// TwinCAT 3 PLC project EngineControlSystem
// ProgramVersion: 3.1.4023.0
// libraries:
//   Tc2_Standard, * (Beckhoff Automation GmbH)
//   Tc2_System, * (Beckhoff Automation GmbH)
//   Tc3_Module, * (Beckhoff Automation GmbH)
//   VisuSymbols,3.5.10.0,System
// project tree:
//   DUTs/ E_RotationDirection.TcDUT, ST_Inputs.TcDUT, ST_Outputs.TcDUT
//   / GlobalTextList.TcGTLO, PlcTask.TcTTO, Visualization Manager.TcVMO (not stored)
//   GVLs/ GVL_Params.TcGVL
//   OLD/ CAN_Example.TcPOU, FB_Encoder_Old1.TcPOU, FB_Encoder_Old2.TcPOU, FB_Encoder_V2.TcPOU, FB_ENCODER_V3.TcPOU, FB_HomingTimer.TcPOU, F_CounterNegativeOverflow.TcPOU (not stored), F_GenerateCANMessage.TcPOU, F_Homing.TcPOU, F_MechToEl.TcPOU, F_VoltageToWord.TcPOU, GVL_Constants.TcGVL, GVL_Measurements.TcGVL
//   POUs/ FB_Controller.TcPOU, FB_CANMessageHandler.TcPOU, FB_Encoder.TcPOU, F_AnalogIntToVoltage.TcPOU, F_VoltageToCurrentConvert.TcPOU, MAIN.TcPOU
//   VISUs/ Visualization.TcVIS
// real-time tasks:
//   TASK PlcTask: cycle T#100us, priority 1, ADS port 350
// I/O:
//   DEVICE Device 2 (EtherCAT), AmsNetId 157.24.88.195.3.1
//     Term 8 (EK1100) [EK1100 EtherCAT Coupler (2A E-Bus)]
//       Term 9 (EL5101-0010) [EL5101-0010 1Ch. Inc. Encoder 5V (20 million increments/s)]
//       Term 10 (EL3702) [EL3702 2Ch. Ana. Input +/-10V, DIFF, Oversample]
//       Term 11 (EL3702) [EL3702 2Ch. Ana. Input +/-10V, DIFF, Oversample]
//       Term 11 (EL6751) [EL6751 CANopen Master]
//       Term 12 (EL9011) [EL9011 End Terminal]
//   DEVICE Device 1 (COM Port)
//   DEVICE Device 3 (EL6751), AmsNetId 157.24.88.195.4.1
//     Zybo (CAN Interface)
// variable links:
//   EngineControlSystem/EngineControlSystem Instance <-> Device 2 (EtherCAT)/Term 8 (EK1100)/Term 10 (EL3702)
//     PlcTask Inputs/MAIN.stInputs.nEL3702Ch1_In <-> Ch1 Sample 0/Ch1 Value
//     PlcTask Inputs/MAIN.stInputs.nEL3702Ch2_In <-> Ch2 Sample 0/Ch2 Value
//   EngineControlSystem/EngineControlSystem Instance <-> Device 2 (EtherCAT)/Term 8 (EK1100)/Term 11 (EL3702)
//     PlcTask Inputs/MAIN.stInputs.nEL3702Ch3_In <-> Ch1 Sample 0/Ch1 Value
//   EngineControlSystem/EngineControlSystem Instance <-> Device 2 (EtherCAT)/Term 8 (EK1100)/Term 9 (EL5101-0010)
//     PlcTask Inputs/MAIN.stInputs.bEL5101_CounterSet <-> ENC Status compact/Status/Set counter done
//     PlcTask Inputs/MAIN.stInputs.bEL5101_LatchValid <-> ENC Status compact/Status/Latch C valid
//     PlcTask Inputs/MAIN.stInputs.nEL5101_Counter <-> ENC Status compact/Counter value
//     PlcTask Inputs/MAIN.stInputs.nEL5101_Frequency <-> ENC Frequency/Frequency value
//     PlcTask Inputs/MAIN.stInputs.nEL5101_LatchValue <-> ENC Status compact/Latch value
//     PlcTask Outputs/MAIN.stOutputs.bEL5101_EnabledLatch <-> ENC Control compact/Control/Enable latch C
//     PlcTask Outputs/MAIN.stOutputs.bEL5101_SetCounter <-> ENC Control compact/Control/Set counter
//   EngineControlSystem/EngineControlSystem Instance <-> Device 3 (EL6751)/Zybo (CAN Interface)
//     PlcTask Inputs/MAIN.stInputs.Inputs <-> Inputs/RxQueue
//     PlcTask Outputs/MAIN.stOutputs.Outputs <-> Outputs/TxQueue
//   EngineControlSystem/EngineControlSystem Instance <-> TcCOM Objects/Object2 (controller_21_1_2022)
//     PlcTask Inputs/MAIN.stInputs.fAlpha_U <-> Output/U_alpha_beta[0]
//     PlcTask Inputs/MAIN.stInputs.fBeta_U <-> Output/U_alpha_beta[1]
//     PlcTask Inputs/MAIN.stInputs.iD <-> Output/I_dq[0]
//     PlcTask Inputs/MAIN.stInputs.iQ <-> Output/I_dq[1]
//     PlcTask Outputs/MAIN.stOutputs.fControlEnable <-> Input/enable
//     PlcTask Outputs/MAIN.stOutputs.fIa <-> Input/i_abc[0]
//     PlcTask Outputs/MAIN.stOutputs.fIb <-> Input/i_abc[1]
//     PlcTask Outputs/MAIN.stOutputs.fIc <-> Input/i_abc[2]
//     PlcTask Outputs/MAIN.stOutputs.fTheta <-> Input/theta_m
//     PlcTask Outputs/MAIN.stOutputs.fWmech <-> Input/w_actual_rad_m
//     PlcTask Outputs/MAIN.stOutputs.fWref <-> Input/w_ref_rpm

CONFIGURATION EngineControlSystem
    RESOURCE PLC ON TwinCAT3
        TASK PlcTask(INTERVAL := T#100us, PRIORITY := 1);
        PROGRAM MAIN WITH PlcTask : MAIN;
    END_RESOURCE
END_CONFIGURATION

// ---- DUTs/E_RotationDirection.TcDUT
{attribute 'qualified_only'}
{attribute 'strict'}
TYPE E_RotationDirection :
(
	NONE,
	EDGE_DETECTED
);
END_TYPE

// ---- DUTs/ST_Inputs.TcDUT
TYPE ST_Inputs :
STRUCT
	// CAN
	Inputs 				AT %I*	: CANRXQUEUESTRUCT_N_1;
	
	// IO
	nEL3702Ch1_In 		AT %I*	: INT;
	nEL3702Ch2_In 		AT %I*	: INT;
	nEL3702Ch3_In 		AT %I*	: INT;
	
	// Encoder
	nEL5101_Counter 	AT %I*	: UINT;
	bEL5101_CounterSet	AT %I*	: BIT;
	nEL5101_LatchValue	AT %I*	: UINT;
	nEL5101_Frequency	AT %I*	: UDINT;
	bEL5101_LatchValid	AT %I*	: BIT;
	
	// From controller
	fAlpha_U, fBeta_U	AT %I*	: LREAL;
	iQ, iD				AT %I*	: LREAL;
END_STRUCT
END_TYPE

// ---- DUTs/ST_Outputs.TcDUT
TYPE ST_Outputs :
STRUCT
	// To controller
	fWref 					AT %Q*				: LREAL;
	fWmech					AT %Q* 				: LREAL;
	fIa, fIb, fIc 			AT %Q*				: LREAL;
	fTheta	 				AT %Q* 				: LREAL;
	fControlEnable 			AT %Q*				: LREAL;
	
	// CAN
	Outputs					AT %Q*				: CANTXQUEUESTRUCT_N_1;
	
	// Encoder
	nEL5101_SetCounterValue AT %Q*				: UINT;
	bEL5101_SetCounter		AT %Q*				: BIT;
	bEL5101_EnabledLatch	AT %Q*				: BIT;
END_STRUCT
END_TYPE

// ---- GVLs/GVL_Params.TcGVL
VAR_GLOBAL CONSTANT
	SS_INITIALIZE: SINT := 0;
	SS_STEP: SINT := 1;
END_VAR

// ---- OLD/GVL_Constants.TcGVL
{attribute 'qualified_only'}
VAR_GLOBAL CONSTANT
	PI 					: REAL 	:= 3.141592654;
	SPEED_CALC_Cycle 	: INT 	:= 100; 			// in microseconds
	NUMBER_OF_POLEPAIRS : UINT 	:= 5;
	PULSES_PER_REV 		: UINT 	:= 4096*4;
END_VAR

// ---- OLD/GVL_Measurements.TcGVL
{attribute 'qualified_only'}
VAR_GLOBAL
	COUNTER_VALUE		: UINT;
	COUNTER_OFFSET    	: UINT := 0;
	homing_done_encoder	: BOOL;
END_VAR

// ---- POUs/MAIN.TcPOU
PROGRAM MAIN
VAR
	// To controller
	bInit									: BOOL;
	fWRefPrep								: LREAL;
	
	fThetaOl								: REAL;
	
	fVa, fVb								: REAL;
	
	bZeroingDone							: BOOL;
	tpIdRun									: TP;
	tpZeroingWaitTime						: TP;
	tZeroingWaitTime						: TIME := T#1S;
	tIdTime									: TIME := T#5S;
	fElZeroAngle							: LREAL;
	
	bControlEnable							: BOOL;
	bStartHoming							: BOOL;
	bOpenLoop 								: BOOL;
	bHomingDone 							: BOOL;
	fHomingVa								: REAL := 0.5;
	fHomingVb								: REAL := 0;
	
	fbCAN_MessageHandler					: FB_CANMessageHandler();
	fbEncoder								: FB_Encoder();
	
	fbController							: FB_Controller();
	
	stInputs								: ST_Inputs;
	stOutputs								: ST_Outputs;
END_VAR

// Calling encoder and getting outputs and giving inputs
fbEncoder(	stInputs	:= stInputs,
			stOutputs	:= stOutputs,
			fThetaMech 	=> stOutputs.fTheta,
			fOmegaMech 	=> stOutputs.fWmech
);

// Id run to zero pulse location aka latch
IF NOT bZeroingDone THEN
	stOutputs.bEL5101_EnabledLatch := TRUE;
	
		fbCAN_MessageHandler(Inputs := stInputs.Inputs, 
							Outputs := stOutputs.Outputs, 
							fVoltage_A := SIN(fThetaOl),
							fVoltage_B := COS(fThetaOl));
		
		fThetaOl := fThetaOl + 2 * LREAL_TO_REAL( PI ) / 2500;
		IF fThetaOl > 2 * PI THEN
			fThetaOl := 0;
		END_IF
	
	IF stInputs.bEL5101_LatchValid THEN
		stOutputs.nEL5101_SetCounterValue := stInputs.nEL5101_LatchValue;
		stOutputs.bEL5101_SetCounter := TRUE;
		bZeroingDone := stInputs.bEL5101_CounterSet;
		stOutputs.bEL5101_EnabledLatch := FALSE;
		bStartHoming := TRUE;
	END_IF
END_IF

tpZeroingWaitTime( IN := bStartHoming, PT := tZeroingWaitTime );

// Homing
IF bStartHoming AND NOT bHomingDone AND NOT tpZeroingWaitTime.Q THEN
	tpIdRun( IN := bStartHoming, PT := tIdTime );
	stOutputs.fControlEnable := 0;
	fbCAN_MessageHandler(Inputs := stInputs.Inputs, 
						Outputs := stOutputs.Outputs, 
						fVoltage_A := fHomingVa,
						fVoltage_B := fHomingVb);
	
	IF NOT tpIdRun.Q THEN
		fElZeroAngle := fbEncoder.fThetaMech;
		bHomingDone := TRUE;
	END_IF
END_IF

// Enabling for old controller
IF bControlEnable THEN
	stOutputs.fControlEnable := 1;
ELSE	
	stOutputs.fControlEnable := 0;
END_IF 

// Getting controller outputs and giving inputs
fbController.speedrefrpm := fWRefPrep;

fbController.anglerad := -1 * ( fbEncoder.fThetaMech - fElZeroAngle );
// Multiplying the mechanical speed with number of pole pairs gives us the electrical field rotation speed
fbController.speedmeasrad := -1 * fbEncoder.fOmegaMech * 2;

fbController.Current_abc[0] := stInputs.nEL3702Ch1_In;
fbController.Current_abc[1] := stInputs.nEL3702Ch2_In;
fbController.Current_abc[2] := stInputs.nEL3702Ch3_In;

// Controller init
IF NOT bInit THEN
	fbController( ssMethodType := SS_INITIALIZE );
	bInit := TRUE;
END_IF

// Scaling of 0.9 used because svpwm doesnt like full 1 and the scaling in controller uses 400 V which is also the saturation point
fVa := LREAL_TO_REAL(fbController.Voltageoutalphabeta[0] * 0.9);
fVb := LREAL_TO_REAL(fbController.Voltageoutalphabeta[1] * 0.9);

// Enabling controller or open loop
IF bHomingDone THEN
	IF bControlEnable THEN
		IF bInit THEN
			fbController( ssMethodType := SS_STEP );
		END_IF
		fbCAN_MessageHandler(Inputs := stInputs.Inputs, 
							Outputs := stOutputs.Outputs, 
							fVoltage_A := fVa,
							fVoltage_B := fVb);
	ELSIF bOpenLoop THEN
		fbCAN_MessageHandler(Inputs := stInputs.Inputs, 
							Outputs := stOutputs.Outputs, 
							fVoltage_A := SIN(fThetaOl),
							fVoltage_B := COS(fThetaOl));
		
		fThetaOl := fThetaOl + 2 * LREAL_TO_REAL( PI ) / 2500;
		IF fThetaOl > 2 * PI THEN
			fThetaOl := 0;
		END_IF
	END_IF
END_IF

END_PROGRAM

// ---- POUs/FB_CANMessageHandler.TcPOU
FUNCTION_BLOCK FB_CANMessageHandler
VAR_INPUT
	Outputs 	: REFERENCE TO CANTXQUEUESTRUCT_N_1; // CAN muuttujat
	Inputs 		: REFERENCE TO CANRXQUEUESTRUCT_N_1;
	
	fVoltage_A	: REAL; // Jännite A realina
	fVoltage_B	: REAL; // Jännite B realina
END_VAR
VAR
	i				: DINT;
	MessageReceived : CANQUEUE;
	MessageToSend	: CANQUEUE;
	NumberOfMessagesToSend	: UINT := 1;
	wV_a,wV_b		: WORD;
END_VAR

wV_a := M_VoltageToWord(Voltage_In := fVoltage_A);
wV_b := M_VoltageToWord(Voltage_In := fVoltage_B);

MessageToSend := M_GenerateCANMessage(cobID := 4, V_a := wV_a, V_b := wV_b);

IF Outputs.TxCounter = Inputs.TxCounter THEN
   	Outputs.TxMessages[0] := MessageToSend;
    Outputs.NoOfTxMessages := NumberOfMessagesToSend;
    Outputs.TxCounter := Outputs.TxCounter + 1;
END_IF

METHOD M_GenerateCANMessage : CANQUEUE
VAR_INPUT
	cobID	: UINT;
	V_a		: WORD;
	V_b		: WORD;
END_VAR
VAR
	i,j 		: UINT;
	Tempdata	: USINT;
	V_DWORD		: WORD;
	tempMessage : CANMESSAGE;
END_VAR

// WIP CAN Message writing.
(*
	Viestiin tulee Va ja Vb (ilmeisesti). Yksi CAN Frame on käytössä näille kahdelle muuttujalle.
	CANQUEUE Objekti on yksi CAN viesti, joka lähetetään COB ID:seen ja se sisältää 8 kpl UINT muuttujia, jotka varmaankin kirjoitetaan sarjassa, josta muodostuu se 64 bittinen CAN Frame.
	Ei kyllä ole kamalasti ideaa että missä järjestyksessä ne kirjoitetaan sinne. Eli pitäisi varmaankin testata. 
	Koodi on nyt silleensä että oletetaan että kirjoitetaan 7 -> 0. Jolloin 7:n data yksikön merkitsevin bitti on koko framen merkisevin
	Vastaavasti 0:n viimeinen bitti on koko framen viimeinen kirjoitettava bitti.
*)


M_GenerateCANMessage.cobId := cobID;

V_DWORD := V_a;
FOR j := 0 TO 1 DO // First part of frame reserved for V_a
	CASE j OF // ST is dumb language and doesnt allow looping for bit access.
		1:
			Tempdata.0 := V_DWORD.0;
			Tempdata.1 := V_DWORD.1;
			Tempdata.2 := V_DWORD.2;
			Tempdata.3 := V_DWORD.3;
			Tempdata.4 := V_DWORD.4;
			Tempdata.5 := V_DWORD.5;
			Tempdata.6 := V_DWORD.6;
			Tempdata.7 := V_DWORD.7;
			
		0:
			Tempdata.0 := V_DWORD.8;
			Tempdata.1 := V_DWORD.9;
			Tempdata.2 := V_DWORD.10;
			Tempdata.3 := V_DWORD.11;
			Tempdata.4 := V_DWORD.12;
			Tempdata.5 := V_DWORD.13;
			Tempdata.6 := V_DWORD.14;
			Tempdata.7 := V_DWORD.15;
	ELSE
		RETURN;
	END_CASE
	M_GenerateCANMessage.data[j] := Tempdata;
END_FOR

V_DWORD := V_b;
FOR j := 2 TO 3 DO // Second part is reserved for V_b
	CASE j OF // ST is dumb language and doesnt allow looping for bit access.
		3:
			Tempdata.0 := V_DWORD.0;
			Tempdata.1 := V_DWORD.1;
			Tempdata.2 := V_DWORD.2;
			Tempdata.3 := V_DWORD.3;
			Tempdata.4 := V_DWORD.4;
			Tempdata.5 := V_DWORD.5;
			Tempdata.6 := V_DWORD.6;
			Tempdata.7 := V_DWORD.7;
			
		2:
			Tempdata.0 := V_DWORD.8;
			Tempdata.1 := V_DWORD.9;
			Tempdata.2 := V_DWORD.10;
			Tempdata.3 := V_DWORD.11;
			Tempdata.4 := V_DWORD.12;
			Tempdata.5 := V_DWORD.13;
			Tempdata.6 := V_DWORD.14;
			Tempdata.7 := V_DWORD.15;
	ELSE
		RETURN;
	END_CASE
	M_GenerateCANMessage.data[j] := Tempdata;
END_FOR
END_METHOD

METHOD M_VoltageToWord : WORD
VAR_INPUT
	Voltage_In			: REAL; // Voltage input
END_VAR
VAR
	VoltageMultiplier	: REAL;
	MaxWordValue		: REAL := 16#FFFF;
	Voltage_High_Value 	: REAL := 0.866;
	Voltage_Low_Value	: REAL := -0.866;
END_VAR
// Check that voltage value is between min and max value.
IF Voltage_In > Voltage_High_Value THEN
	Voltage_In := Voltage_High_Value;
ELSIF Voltage_In < Voltage_Low_Value THEN
	Voltage_In := Voltage_Low_Value;
END_IF

VoltageMultiplier := (Voltage_In-Voltage_Low_Value)/(Voltage_High_Value-Voltage_Low_Value);

M_VoltageToWord := UINT_TO_WORD(REAL_TO_UINT(VoltageMultiplier*MaxWordValue));
END_METHOD

END_FUNCTION_BLOCK

// ---- POUs/FB_Encoder.TcPOU
FUNCTION_BLOCK FB_Encoder
VAR_INPUT
	stInputs				: REFERENCE TO ST_Inputs;
	stOutputs				: REFERENCE TO ST_Outputs;
END_VAR
VAR_OUTPUT
	fThetaMech				: LREAL;
	fOmegaMech				: LREAL;
END_VAR
VAR
	bUseLatch				: BOOL;
	bInit					: BOOL;
	fOmegaMechNoDirection	: LREAL := 0.0; // No rotation direction
	fRotationDirection		: LREAL := 0.0;
	fPpr					: LREAL := 4096;
	fFreqScale				: LREAL := 0.01;
	f16bitMax				: LREAL := 65535;
	nCounter				: UINT;
	fTheta					: LREAL := 0.0;
	fThetaPrev				: LREAL := 0.0;
	nThetaDelta				: LREAL := 0.0;
	nThetaDeltaPrev			: LREAL := 0.0;
END_VAR



// Angle calculation
nCounter		:= stInputs.nEL5101_Counter * 4;
fThetaPrev 		:= fTheta;
fTheta	:= ( 2.0 * PI ) - ( UINT_TO_LREAL( nCounter ) / f16bitMax * 2.0 * PI ); // Counter is divided by max value of UINT times two because one circle is 2pi


// Rotation direction calculation
IF bUseLatch THEN
	stOutputs.bEL5101_EnabledLatch := TRUE;
	
	IF stInputs.nEL5101_LatchValue < stInputs.nEL5101_Counter THEN
		fRotationDirection := -1;
	ELSIF stInputs.nEL5101_LatchValue > stInputs.nEL5101_Counter THEN
		fRotationDirection := 1;
	END_IF
	
	stOutputs.bEL5101_EnabledLatch := FALSE;
	
ELSE
	nThetaDeltaPrev := nThetaDelta;
	nThetaDelta		:= fTheta - fThetaPrev;
	
	IF nThetaDelta < 0 AND nThetaDeltaPrev < 0 THEN
		fRotationDirection := 1;
	ELSIF  nThetaDelta > 0 AND nThetaDeltaPrev > 0  THEN
			fRotationDirection := -1;
	END_IF
END_IF

// Angle speed calculation
fOmegaMechNoDirection := 2.0 * PI * ( UDINT_TO_LREAL( stInputs.nEL5101_Frequency ) / fPpr * fFreqScale );

// Outputs
fThetaMech	:= fTheta;
fOmegaMech 	:= fRotationDirection * fOmegaMechNoDirection;

END_FUNCTION_BLOCK

// ---- POUs/FB_Controller.TcPOU
FUNCTION_BLOCK FB_Controller
VAR_INPUT
	ssMethodType: SINT;
	speedrefrpm: LREAL;
	Current_abc: ARRAY[0..2] OF LREAL;
	speedmeasrad: LREAL;
	anglerad: LREAL;
END_VAR
VAR_OUTPUT
	Voltageoutalphabeta: ARRAY[0..1] OF LREAL;
	Electrictorguecommand: LREAL;
	Currentmeasalphabeta: ARRAY[0..1] OF LREAL;
	Currentmeasdq: ARRAY[0..1] OF LREAL;
	Currentcommanddq: ARRAY[0..1] OF LREAL;
	Voltagecommanddq: ARRAY[0..1] OF LREAL;
	Voltagecommandalphabeta: ARRAY[0..1] OF LREAL;
END_VAR
VAR
	rtb_IntegralGain: LREAL;
	rtb_DeadZone: LREAL;
	rtb_DeadZone_p: LREAL;
	rtb_idref: LREAL;
	rtb_Gain3: LREAL;
	rtb_IntegralGain_p: LREAL;
	rtb_Gain4: LREAL;
	rtb_Fcn: LREAL;
	rtb_Integrator_k: LREAL;
	rtb_Fcn1: LREAL;
	rtb_iqref: LREAL;
	rtb_IntegralGain_h: LREAL;
	rtb_DeadZone_c: LREAL;
	rtb_Saturation: LREAL;
	rtb_Switch2: SINT;
	rtb_Switch1: SINT;
	rtb_Saturation_h_idx_0: LREAL;
	rtb_Saturation_h_idx_1: LREAL;
	temp1: LREAL;
	Gain3: LREAL;
	Integrator_DSTATE: LREAL;
	Integrator_DSTATE_c: LREAL;
	Integrator_DSTATE_m: LREAL;
	Gain2: LREAL;
	Sqrt2: LREAL;
	Gain4: LREAL;
END_VAR



CASE ssMethodType OF
    SS_INITIALIZE: 
        (* SystemInitialize for Atomic SubSystem: '<Root>/Controller_subsystem_29112022' *)
        (* InitializeConditions for DiscreteIntegrator: '<S145>/Integrator' *)
        Integrator_DSTATE := 0.0;
        (* InitializeConditions for DiscreteIntegrator: '<S43>/Integrator' *)
        Integrator_DSTATE_c := 0.0;
        (* InitializeConditions for DiscreteIntegrator: '<S93>/Integrator' *)
        Integrator_DSTATE_m := 0.0;
        (* End of SystemInitialize for SubSystem: '<Root>/Controller_subsystem_29112022' *)
        

        (* ConstCode for Atomic SubSystem: '<Root>/Controller_subsystem_29112022' *)
        (* ConstCode for Gain: '<S3>/Gain2' incorporates:
         *  Constant: '<S3>/Constant' *)
        Gain2 := 2.1427199999999997;
        (* ConstCode for Sqrt: '<S3>/Sqrt2' incorporates:
         *  Constant: '<S3>/Constant1' *)
        Sqrt2 := 1.4142135623730951;
        (* ConstCode for Gain: '<S3>/Gain3' *)
        Gain3 := 0.44739 * Sqrt2;
        (* ConstCode for Gain: '<S3>/Gain4' incorporates:
         *  Constant: '<S3>/Constant2' *)
        Gain4 := 2.1427199999999997;
        (* End of ConstCode for SubSystem: '<Root>/Controller_subsystem_29112022' *)
    SS_STEP: 
        (* Outputs for Atomic SubSystem: '<Root>/Controller_subsystem_29112022' *)
        (* Sum: '<S4>/Add1' incorporates:
         *  Gain: '<S1>/toRad' *)
        rtb_IntegralGain := (0.10471975511965977 * speedrefrpm) - speedmeasrad;
        (* Sum: '<S154>/Sum' incorporates:
         *  DiscreteIntegrator: '<S145>/Integrator'
         *  Gain: '<S150>/Proportional Gain' *)
        rtb_DeadZone := (0.1 * rtb_IntegralGain) + Integrator_DSTATE;
        (* Saturate: '<S152>/Saturation' *)

        IF rtb_DeadZone > 7.0 THEN 
            rtb_DeadZone_p := 7.0;
        ELSIF rtb_DeadZone >= -7.0 THEN 
            rtb_DeadZone_p := rtb_DeadZone;
        ELSE 
            rtb_DeadZone_p := -7.0;
        END_IF;

        (* End of Saturate: '<S152>/Saturation' *)
        

        (* Switch: '<S4>/Switch' incorporates:
         *  Constant: '<S4>/Constant3' *)

        IF rtb_DeadZone_p <> 0.0 THEN 
            Electrictorguecommand := rtb_DeadZone_p;
        ELSE 
            Electrictorguecommand := 0.01;
        END_IF;

        (* End of Switch: '<S4>/Switch' *)
        

        (* Product: '<S3>/Divide1' incorporates:
         *  Abs: '<S3>/Abs'
         *  Gain: '<S3>/Gain1'
         *  Product: '<S3>/Divide'
         *  Sqrt: '<S3>/Sqrt1' *)
        temp1 := ABS(Electrictorguecommand);
        rtb_idref := SQRT((0.1615435812 * temp1) / Gain2) / Gain3;
        (* Gain: '<S5>/Gain3' incorporates:
         *  Gain: '<S5>/Gain1'
         *  Gain: '<S5>/Gain2'
         *  Sum: '<S5>/Sum' *)
        rtb_Gain3 := (((-0.5 * Current_abc[1]) + Current_abc[0]) + (-0.5 * Current_abc[2])) * 0.66666666666666663;
        (* Gain: '<S5>/Gain4' incorporates:
         *  Gain: '<S5>/Gain6'
         *  Gain: '<S5>/Gain7'
         *  Sum: '<S5>/Sum1' *)
        rtb_Gain4 := ((0.8660254037844386 * Current_abc[1]) + (-0.8660254037844386 * Current_abc[2])) * 0.66666666666666663;
        (* Fcn: '<S6>/Fcn' incorporates:
         *  Fcn: '<S6>/Fcn1'
         *  Fcn: '<S7>/Fcn'
         *  Fcn: '<S7>/Fcn1' *)
        rtb_Saturation_h_idx_0 := SIN(anglerad);
        rtb_Saturation_h_idx_1 := COS(anglerad);
        rtb_Fcn := (rtb_Gain3 * rtb_Saturation_h_idx_1) + (rtb_Gain4 * rtb_Saturation_h_idx_0);
        (* Sum: '<S2>/Add' *)
        rtb_IntegralGain_p := rtb_idref - rtb_Fcn;
        (* Sum: '<S52>/Sum' incorporates:
         *  DiscreteIntegrator: '<S43>/Integrator'
         *  Gain: '<S48>/Proportional Gain' *)
        rtb_DeadZone_p := (2.0 * rtb_IntegralGain_p) + Integrator_DSTATE_c;
        (* Saturate: '<S50>/Saturation' *)

        IF rtb_DeadZone_p > 400.0 THEN 
            rtb_Integrator_k := 400.0;
        ELSIF rtb_DeadZone_p >= -400.0 THEN 
            rtb_Integrator_k := rtb_DeadZone_p;
        ELSE 
            rtb_Integrator_k := -400.0;
        END_IF;

        (* End of Saturate: '<S50>/Saturation' *)
        

        (* Fcn: '<S6>/Fcn1' *)
        rtb_Fcn1 := (( -rtb_Gain3) * rtb_Saturation_h_idx_0) + (rtb_Gain4 * rtb_Saturation_h_idx_1);
        (* Product: '<S3>/Divide2' incorporates:
         *  Gain: '<S3>/Gain5'
         *  Product: '<S3>/Multiply' *)
        rtb_iqref := (2.0 * Electrictorguecommand) / (Gain4 * rtb_idref);
        (* Sum: '<S2>/Add1' *)
        rtb_IntegralGain_h := rtb_iqref - rtb_Fcn1;
        (* Sum: '<S2>/Add2' incorporates:
         *  Gain: '<S2>/Gain'
         *  Product: '<S2>/Product' *)
        rtb_Integrator_k := rtb_Integrator_k - ((0.09027 * rtb_Fcn1) * speedmeasrad);
        (* Sum: '<S102>/Sum' incorporates:
         *  DiscreteIntegrator: '<S93>/Integrator'
         *  Gain: '<S98>/Proportional Gain' *)
        rtb_DeadZone_c := (2.0 * rtb_IntegralGain_h) + Integrator_DSTATE_m;
        (* Saturate: '<S100>/Saturation' *)

        IF rtb_DeadZone_c > 400.0 THEN 
            rtb_Saturation := 400.0;
        ELSIF rtb_DeadZone_c >= -400.0 THEN 
            rtb_Saturation := rtb_DeadZone_c;
        ELSE 
            rtb_Saturation := -400.0;
        END_IF;

        (* End of Saturate: '<S100>/Saturation' *)
        

        (* Sum: '<S2>/Add3' incorporates:
         *  Gain: '<S2>/Gain1'
         *  Product: '<S2>/Product1' *)
        rtb_Saturation := ((0.44739 * rtb_Fcn) * speedmeasrad) + rtb_Saturation;
        (* Saturate: '<S1>/Saturation' incorporates:
         *  Fcn: '<S7>/Fcn'
         *  Fcn: '<S7>/Fcn1'
         *  Outport: '<Root>/Voltage command alpha-beta' *)
        Voltagecommandalphabeta[0] := (rtb_Integrator_k * rtb_Saturation_h_idx_1) - (rtb_Saturation * rtb_Saturation_h_idx_0);
        Voltagecommandalphabeta[1] := (rtb_Integrator_k * rtb_Saturation_h_idx_0) + (rtb_Saturation * rtb_Saturation_h_idx_1);

        IF Voltagecommandalphabeta[0] > 400.0 THEN 
            rtb_Saturation_h_idx_0 := 400.0;
        ELSIF Voltagecommandalphabeta[0] >= -400.0 THEN 
            rtb_Saturation_h_idx_0 := Voltagecommandalphabeta[0];
        ELSE 
            rtb_Saturation_h_idx_0 := -400.0;
        END_IF;


        IF Voltagecommandalphabeta[1] > 400.0 THEN 
            rtb_Saturation_h_idx_1 := 400.0;
        ELSIF Voltagecommandalphabeta[1] >= -400.0 THEN 
            rtb_Saturation_h_idx_1 := Voltagecommandalphabeta[1];
        ELSE 
            rtb_Saturation_h_idx_1 := -400.0;
        END_IF;

        (* End of Saturate: '<S1>/Saturation' *)
        

        (* DeadZone: '<S36>/DeadZone' *)

        IF rtb_DeadZone_p > 400.0 THEN 
            rtb_DeadZone_p := rtb_DeadZone_p - 400.0;
            (* Switch: '<S34>/Switch1' incorporates:
             *  Constant: '<S34>/Constant' *)
            rtb_Switch2 := 1;
        ELSE 

            IF rtb_DeadZone_p >= -400.0 THEN 
                rtb_DeadZone_p := 0.0;
            ELSE 
                rtb_DeadZone_p := rtb_DeadZone_p - -400.0;
            END_IF;

            (* Switch: '<S34>/Switch1' incorporates:
             *  Constant: '<S34>/Constant2' *)
            rtb_Switch2 := -1;
        END_IF;

        (* End of DeadZone: '<S36>/DeadZone' *)
        

        (* Gain: '<S40>/Integral Gain' *)
        rtb_IntegralGain_p := 0.2 * rtb_IntegralGain_p;
        (* Switch: '<S34>/Switch2' incorporates:
         *  Constant: '<S34>/Clamping_zero'
         *  Constant: '<S34>/Constant3'
         *  Constant: '<S34>/Constant4'
         *  RelationalOperator: '<S34>/fix for DT propagation issue1' *)

        IF rtb_IntegralGain_p > 0.0 THEN 
            rtb_Switch1 := 1;
        ELSE 
            rtb_Switch1 := -1;
        END_IF;

        (* End of Switch: '<S34>/Switch2' *)
        

        (* Switch: '<S34>/Switch' incorporates:
         *  Constant: '<S34>/Clamping_zero'
         *  Constant: '<S34>/Constant1'
         *  Logic: '<S34>/AND3'
         *  RelationalOperator: '<S34>/Equal1'
         *  RelationalOperator: '<S34>/Relational Operator' *)

        IF (rtb_DeadZone_p <> 0.0) AND (rtb_Switch2 = rtb_Switch1) THEN 
            rtb_IntegralGain_p := 0.0;
        END_IF;

        (* End of Switch: '<S34>/Switch' *)
        

        (* DeadZone: '<S86>/DeadZone' *)

        IF rtb_DeadZone_c > 400.0 THEN 
            rtb_DeadZone_c := rtb_DeadZone_c - 400.0;
            (* Switch: '<S84>/Switch1' incorporates:
             *  Constant: '<S84>/Constant' *)
            rtb_Switch1 := 1;
        ELSE 

            IF rtb_DeadZone_c >= -400.0 THEN 
                rtb_DeadZone_c := 0.0;
            ELSE 
                rtb_DeadZone_c := rtb_DeadZone_c - -400.0;
            END_IF;

            (* Switch: '<S84>/Switch1' incorporates:
             *  Constant: '<S84>/Constant2' *)
            rtb_Switch1 := -1;
        END_IF;

        (* End of DeadZone: '<S86>/DeadZone' *)
        

        (* Gain: '<S90>/Integral Gain' *)
        rtb_IntegralGain_h := 0.2 * rtb_IntegralGain_h;
        (* Switch: '<S84>/Switch2' incorporates:
         *  Constant: '<S84>/Clamping_zero'
         *  Constant: '<S84>/Constant3'
         *  Constant: '<S84>/Constant4'
         *  RelationalOperator: '<S84>/fix for DT propagation issue1' *)

        IF rtb_IntegralGain_h > 0.0 THEN 
            rtb_Switch2 := 1;
        ELSE 
            rtb_Switch2 := -1;
        END_IF;

        (* End of Switch: '<S84>/Switch2' *)
        

        (* Switch: '<S84>/Switch' incorporates:
         *  Constant: '<S84>/Clamping_zero'
         *  Constant: '<S84>/Constant1'
         *  Logic: '<S84>/AND3'
         *  RelationalOperator: '<S84>/Equal1'
         *  RelationalOperator: '<S84>/Relational Operator' *)

        IF (rtb_DeadZone_c <> 0.0) AND (rtb_Switch1 = rtb_Switch2) THEN 
            rtb_IntegralGain_h := 0.0;
        END_IF;

        (* End of Switch: '<S84>/Switch' *)
        

        (* DeadZone: '<S138>/DeadZone' *)

        IF rtb_DeadZone > 7.0 THEN 
            rtb_DeadZone := rtb_DeadZone - 7.0;
            (* Switch: '<S136>/Switch1' incorporates:
             *  Constant: '<S136>/Constant' *)
            rtb_Switch1 := 1;
        ELSE 

            IF rtb_DeadZone >= -7.0 THEN 
                rtb_DeadZone := 0.0;
            ELSE 
                rtb_DeadZone := rtb_DeadZone - -7.0;
            END_IF;

            (* Switch: '<S136>/Switch1' incorporates:
             *  Constant: '<S136>/Constant2' *)
            rtb_Switch1 := -1;
        END_IF;

        (* End of DeadZone: '<S138>/DeadZone' *)
        

        (* Gain: '<S142>/Integral Gain' *)
        rtb_IntegralGain := 0.05 * rtb_IntegralGain;
        (* Switch: '<S136>/Switch2' incorporates:
         *  Constant: '<S136>/Clamping_zero'
         *  Constant: '<S136>/Constant3'
         *  Constant: '<S136>/Constant4'
         *  RelationalOperator: '<S136>/fix for DT propagation issue1' *)

        IF rtb_IntegralGain > 0.0 THEN 
            rtb_Switch2 := 1;
        ELSE 
            rtb_Switch2 := -1;
        END_IF;

        (* End of Switch: '<S136>/Switch2' *)
        

        (* Switch: '<S136>/Switch' incorporates:
         *  Constant: '<S136>/Clamping_zero'
         *  Constant: '<S136>/Constant1'
         *  Logic: '<S136>/AND3'
         *  RelationalOperator: '<S136>/Equal1'
         *  RelationalOperator: '<S136>/Relational Operator' *)

        IF (rtb_DeadZone <> 0.0) AND (rtb_Switch1 = rtb_Switch2) THEN 
            rtb_IntegralGain := 0.0;
        END_IF;

        (* End of Switch: '<S136>/Switch' *)
        

        (* Update for DiscreteIntegrator: '<S145>/Integrator' *)
        Integrator_DSTATE := (5.0E-5 * rtb_IntegralGain) + Integrator_DSTATE;
        (* Update for DiscreteIntegrator: '<S43>/Integrator' *)
        Integrator_DSTATE_c := (5.0E-5 * rtb_IntegralGain_p) + Integrator_DSTATE_c;
        (* Update for DiscreteIntegrator: '<S93>/Integrator' *)
        Integrator_DSTATE_m := (5.0E-5 * rtb_IntegralGain_h) + Integrator_DSTATE_m;
        (* Outport: '<Root>/Voltage out alpha-beta' incorporates:
         *  Gain: '<S1>/normalize' *)
        Voltageoutalphabeta[0] := 0.0025 * rtb_Saturation_h_idx_0;
        Voltageoutalphabeta[1] := 0.0025 * rtb_Saturation_h_idx_1;
        (* End of Outputs for SubSystem: '<Root>/Controller_subsystem_29112022' *)
        

        (* Outport: '<Root>/Current meas alpha-beta' *)
        Currentmeasalphabeta[0] := rtb_Gain3;
        Currentmeasalphabeta[1] := rtb_Gain4;
        (* Outport: '<Root>/Current meas dq' *)
        Currentmeasdq[0] := rtb_Fcn;
        Currentmeasdq[1] := rtb_Fcn1;
        (* Outport: '<Root>/Current command dq' *)
        Currentcommanddq[0] := rtb_idref;
        Currentcommanddq[1] := rtb_iqref;
        (* Outport: '<Root>/Voltage command dq' *)
        Voltagecommanddq[0] := rtb_Integrator_k;
        Voltagecommanddq[1] := rtb_Saturation;
END_CASE;

END_FUNCTION_BLOCK

// ---- OLD/CAN_Example.TcPOU
FUNCTION_BLOCK CAN_Example
VAR_INPUT
END_VAR
VAR_OUTPUT
END_VAR
VAR
	fPhase1_Uptime	: DINT;
	fPhase2_Uptime	: DINT;
	fPhase3_Uptime	: DINT;
	fPhase1_Offset	: DINT;
	fPhase2_Offset	: DINT;
	fPhase3_Offset	: DINT;
END_VAR

(*
Example codes from some beckhoff PDF

Sample code: Sending messages from the PLC
if Outputs.TxCounter = Inputs.TxCounter then
          for i=0 to NumberOfMessagesToSend do
                  Outputs.TxMessage[i] = MessageToSend[i];
          End_for
          Outputs.NoOfTxMessages = NumberOfMessagesToSend;
          Outputs.TxCounter := Outputs.TxCounter + 1;
end_if


Sample code: Receiving messages from the PLC
if Outputs.RxCounter <> Inputs.RxCounter then
          for I := 0 to (Inputs.NoOfRxMessages-1) do
                   MessageReceived[i] := Inputs.RxMessage [i];
          End_for
          Outputs.RxCounter := Outputs.RxCounter+1;
end_if

*)

END_FUNCTION_BLOCK

// ---- OLD/FB_Encoder_Old1.TcPOU
FUNCTION_BLOCK FB_Encoder_Old1
VAR_OUTPUT
	THETA 					: REAL;
	THETA_EL 				: REAL;
	OMEGA					: REAL;
END_VAR
VAR
	OMEGA_raw				: REAL;
	OMEGA_filtered			: REAL;
	Omega_prev				: REAL;
	THETA_rads				: REAL;
	THETA_prev_rads			: REAL;
	
	THETA_PREV 				: REAL 	:= 0;
	T_S 					: REAL 	:= 0.0001;
	OVERFLOW_SET 			: BOOL 	:= FALSE;
	UNDERFLOW_SET 			: BOOL 	:= FALSE;

	UNDERFLOW_VALUE 		: UINT 	:= 0;
	OVERFLOW_VALUE 			: UINT 	:= 4096*4; //65535;
	DOWNCOUNT_VALUE 		: UINT 	:= 1003;
	UPCOUNT_VALUE 			: UINT 	:= DOWNCOUNT_VALUE + (Constants.PULSES_PER_REV - 1);
	
	INIT_DONE 				: BOOL 	:= FALSE;
	
	COUNTER_VALUE			: UINT;
	I 						: INT 	:= 0;
	COUNTER_VALUE_PREV 		: UINT 	:= Measurements.COUNTER_VALUE;
	COUNTER_OUT 			: UINT 	:= 0;
	FIRSTCYCLE_DONE 		: BOOL 	:= FALSE;
	CLOCKWISE				: BOOL;
	COUNTERCLOCKWISE		: BOOL;
	PLUSONEPULSE 			: BOOL;
	PLUSTWOPULSES 			: BOOL;
	PLUSTHREEPULSES 		: BOOL;
	
	THETA_EST_TOT 			: REAL;
	THETA_EST_TOT_OLD		: REAL	:=0.0;
	THETA_ERR_FAST			: REAL;
	THETA_ERR_HYS			: REAL	:= 0.1;	//0.1
	OMEGA_FAST 				: REAL;
	OMEGA_EST_TOT 			: REAL;
	Ts_EST 					: REAL 	:=1E-4;	//1E-2
	THETA_EST_FAST 			: REAL;
	THETA_EST_FAST_OLD 		: REAL;
	GAIN_EST 				: REAL 	:=20; 	//1
	
	THETA_n 				: REAL; 
	DELTA_THETA_n0 			: REAL :=0.0;
	DELTA_THETA_n1 			: REAL :=0.0; 
	DELTA_THETA 			: REAL;
	temp					: REAL; 
END_VAR

// counter resetointi. kirjoita arvo enc control compact/control/set counter value ja rising edge /control/set counter


COUNTER_VALUE := Measurements.COUNTER_VALUE;

//Init procedure
IF FIRSTCYCLE_DONE = FALSE THEN
(*	STARTING_VALUE := COUNTER_VALUE;
	UP_VALUE := STARTING_VALUE + PULSES_PER_REV;
	DOWN_VALUE := STARTING_VALUE - PULSES_PER_REV;
*)	FIRSTCYCLE_DONE := TRUE;
END_IF

//End of init procedure

//Rotation direction estimation											//ADDED ROTATION  DIRECTION ESTIMATION - FEDOR POLUNIN 07 06 17

	IF (COUNTER_VALUE < COUNTER_VALUE_PREV AND COUNTER_VALUE <= (UNDERFLOW_VALUE + 2) AND COUNTER_VALUE_PREV >= (OVERFLOW_VALUE - 2)) THEN
		CLOCKWISE := TRUE;
		COUNTERCLOCKWISE := FALSE;
	ELSIF (COUNTER_VALUE > COUNTER_VALUE_PREV AND COUNTER_VALUE_PREV <= (UNDERFLOW_VALUE + 2) AND COUNTER_VALUE >= (OVERFLOW_VALUE - 2)) THEN
		COUNTERCLOCKWISE := TRUE;
		CLOCKWISE := FALSE;
	ELSIF 	(COUNTER_VALUE > COUNTER_VALUE_PREV AND COUNTER_VALUE <> OVERFLOW_VALUE) THEN 
		CLOCKWISE := TRUE;
		COUNTERCLOCKWISE := FALSE;
	ELSIF 	(COUNTER_VALUE < COUNTER_VALUE_PREV AND COUNTER_VALUE <> UNDERFLOW_VALUE) THEN
		COUNTERCLOCKWISE := TRUE;
		CLOCKWISE := FALSE;
	END_IF

//COUNTERCLOCKWISE := TRUE;
//CLOCKWISE := TRUE;

//End of Rotation direction estimation 

// Counter value conversion from 0..65535 to DOWNCOUNT_VALUE .. UPCOUNT_VALUE (1003..2002)  		//up to 1200 rpm both directions, no pulse loss w/o load Fedor Polunin 26 06 2017

IF (COUNTER_VALUE <= (UNDERFLOW_VALUE + 2) AND COUNTER_VALUE_PREV >= (OVERFLOW_VALUE - 2)) THEN
	COUNTER_OUT := COUNTER_OUT + (COUNTER_VALUE-UNDERFLOW_VALUE) + (OVERFLOW_VALUE-COUNTER_VALUE_PREV) + 1; 	//added + 1 because otherwise when COUNTER_VALUE resets from 65535 to 0, COUNTER_OUT does not increment
ELSIF (COUNTER_VALUE >= (OVERFLOW_VALUE - 2) AND COUNTER_VALUE_PREV <= (UNDERFLOW_VALUE + 2)) THEN
	COUNTER_OUT := COUNTER_OUT - (OVERFLOW_VALUE-COUNTER_VALUE) - (COUNTER_VALUE_PREV-UNDERFLOW_VALUE) - 1;		//added - 1 because otherwise when COUNTER_VALUE resets from 0 to 65535, COUNTER_OUT does not decrement
ELSIF (COUNTER_VALUE = COUNTER_VALUE_PREV + 1) OR (COUNTER_VALUE = COUNTER_VALUE_PREV + 2) OR (COUNTER_VALUE = COUNTER_VALUE_PREV + 3)THEN			
	COUNTER_OUT := COUNTER_OUT + (COUNTER_VALUE - COUNTER_VALUE_PREV); // + 1;
ELSIF  (COUNTER_VALUE = COUNTER_VALUE_PREV - 1) OR (COUNTER_VALUE = COUNTER_VALUE_PREV - 2) OR (COUNTER_VALUE = COUNTER_VALUE_PREV - 3) THEN; 
	COUNTER_OUT := COUNTER_OUT - (COUNTER_VALUE_PREV - COUNTER_VALUE);//- 1;
END_IF

IF COUNTER_OUT < DOWNCOUNT_VALUE THEN
	COUNTER_OUT := UPCOUNT_VALUE - (DOWNCOUNT_VALUE - COUNTER_OUT) + 1;  // +1 TO PREVENT COUNTER_OUT FROM SETTING UP TO 2001 INSTEAD OF 2002 WHEN DOWNCOUNT_VALUE - COUNTER_OUT = 1
	UNDERFLOW_SET := TRUE;
	
ELSIF COUNTER_OUT > UPCOUNT_VALUE THEN
	COUNTER_OUT := DOWNCOUNT_VALUE + (COUNTER_OUT - UPCOUNT_VALUE) - 1;  //FOR THE SAME REASON
	OVERFLOW_SET := TRUE;
END_IF

(*	
	//Encoder pulses per program cycle counter														
IF (COUNTER_VALUE = COUNTER_VALUE_PREV + 1) THEN
	PLUSONEPULSE := TRUE;
	PLUSTWOPULSES := FALSE;
	PLUSTHREEPULSES := FALSE;
	
ELSIF (COUNTER_VALUE = COUNTER_VALUE_PREV + 2) THEN
	PLUSONEPULSE := FALSE;
	PLUSTWOPULSES := TRUE;
	PLUSTHREEPULSES := FALSE;
	
ELSIF (COUNTER_VALUE = COUNTER_VALUE_PREV + 3) THEN
	PLUSONEPULSE := FALSE;
	PLUSTWOPULSES := FALSE;
	PLUSTHREEPULSES := TRUE;
END_IF
*)

COUNTER_VALUE_PREV := COUNTER_VALUE;

//End of counter value conversion 

// Convert to rotor angle theta in degrees

	THETA := 360.0*INT_TO_REAL(UINT_TO_INT(COUNTER_OUT - DOWNCOUNT_VALUE))/(UPCOUNT_VALUE-DOWNCOUNT_VALUE);		// COUNTER_OUT - DOWNCOUNT_VALUE can be negative, requires INT_TO_REAL 
	IF Measurements.homing_done_encoder THEN
		THETA := 360.0*INT_TO_REAL(COUNTER_OUT - DOWNCOUNT_VALUE)/(UPCOUNT_VALUE-DOWNCOUNT_VALUE) - Measurements.theta_nolla*180/PI;		// COUNTER_OUT - DOWNCOUNT_VALUE can be negative, requires INT_TO_REAL 
		IF THETA < 0 THEN
			temp := Measurements.theta_nolla*180/PI - (360.0*INT_TO_REAL(COUNTER_OUT - DOWNCOUNT_VALUE)/(UPCOUNT_VALUE-DOWNCOUNT_VALUE));
			THETA := 2*PI - temp;
		END_IF
	END_IF
    THETA_EL := 360.0*INT_TO_REAL(((COUNTER_OUT - DOWNCOUNT_VALUE) MOD 200))/200.0;

//End of conversion to rotor angle theta in degrees

//Angular rotation speed omega estimation (in rad/s)
I := I+1;

	THETA_rads := THETA/180*PI;

IF I = Constants.SPEED_CALC_Cycle THEN															
	// Calculate angular speed
		//raw speed estimation algorithm based on backward Euler differentiation
	IF OVERFLOW_SET = TRUE AND THETA < 20 THEN								//Fedor Polunin 06.06.17 - added AND THETA < 10 to prevent this from executing if theta hasn't yet changed from 2pi to zero
		OMEGA := (THETA + (360.0 - THETA_PREV))/(T_S*Constants.SPEED_CALC_Cycle);				
	ELSIF UNDERFLOW_SET = TRUE AND THETA > 340 THEN							//Fedor Polunin 06.06.17 - added AND THETA < 10 to prevent this from executing if theta hasn't yet changed from zero to 2pi
		OMEGA := -((360.0-THETA) + THETA_PREV)/(T_S*Constants.SPEED_CALC_Cycle);					
	ELSE
		IF CLOCKWISE = TRUE AND THETA_PREV > 180 AND THETA < 180 THEN		//Fedor Polunin 06.06.17 - added                                                                                           (IF THETA_PREV > 180 AND THETA < 180 THEN) BUT NOT VALID if both directions are used (it is to ensure correct omega estimation during THETA 2pi to 0 change)
			OMEGA := (THETA + (360.0 - THETA_PREV))/(T_S*Constants.SPEED_CALC_Cycle);			//Fedor Polunin 06.06.17 - added OMEGA := (THETA + (360.0 - THETA_PREV))/(T_S*100.0);
		ELSIF  COUNTERCLOCKWISE = TRUE AND  THETA_PREV < 180 AND THETA > 180 THEN							
			OMEGA := -((360.0-THETA) + THETA_PREV)/(T_S*Constants.SPEED_CALC_Cycle);			
		ELSE																//Fedor Polunin 06.06.17 - ELSE use theta and theta_prev without modification:
			OMEGA := (THETA - THETA_PREV)/(T_S*Constants.SPEED_CALC_Cycle);
		END_IF
	END_IF	
	
	OMEGA_raw := PI*OMEGA/180.0;
	
	//end of raw speed estimation algorithm														
	
	//filtered speed estimation algorithm based on ZOH differentiation + filter + output median filtering		
	IF OVERFLOW_SET = TRUE AND THETA < 20 THEN								//Fedor Polunin 06.06.17 - added AND THETA < 10 to prevent this from executing if theta hasn't yet changed from 2pi to zero
		DELTA_THETA := (THETA_rads + (2*PI - THETA_prev_rads));		
	ELSIF UNDERFLOW_SET = TRUE AND THETA > 340 THEN							//Fedor Polunin 06.06.17 - added AND THETA < 10 to prevent this from executing if theta hasn't yet changed from zero to 2pi
		DELTA_THETA := -((2*PI-THETA_rads ) + THETA_prev_rads);				
	ELSE
		IF CLOCKWISE = TRUE AND THETA_PREV > 180 AND THETA < 180 THEN		//Fedor Polunin 06.06.17 - added                                                                                           (IF THETA_PREV > 180 AND THETA < 180 THEN) BUT NOT VALID if both directions are used (it is to ensure correct omega estimation during THETA 2pi to 0 change)
			DELTA_THETA := (THETA_rads  + (2*PI - THETA_prev_rads));				//Fedor Polunin 06.06.17 - added OMEGA := (THETA + (360.0 - THETA_PREV))/(T_S*100.0);
		ELSIF  COUNTERCLOCKWISE = TRUE AND  THETA_PREV < 180 AND THETA > 180 THEN							
			DELTA_THETA := -((2*PI-THETA_rads ) + THETA_prev_rads);	
		ELSE																//Fedor Polunin 06.06.17 - ELSE use theta and theta_prev without modification:
			DELTA_THETA := (THETA_rads  - THETA_prev_rads);	
		END_IF
	END_IF														
	
	DELTA_THETA_n0:=0.5*DELTA_THETA+ 0.5*DELTA_THETA_n1;
 	DELTA_THETA_n1:= DELTA_THETA_n0;
	OMEGA_filtered := DELTA_THETA_n0*33*104.0166/21.23 +  0.189 * Omega_prev ;	

	THETA_PREV := THETA;
	THETA_prev_rads := THETA_rads;
	OMEGA_prev:= OMEGA_filtered;
	
	//end of filtered speed estimation algorithm
	
	I := 0;

	UNDERFLOW_SET := FALSE;
	OVERFLOW_SET := FALSE;
	
	//Speed feedback signal selection
		//OMEGA:=OMEGA_raw;
		OMEGA:=OMEGA_filtered;
		//OMEGA := PI*OMEGA/180.0;
END_IF;
	
	//fast speed estimator part (filtered algorithm above is the slow part) - refer to the paper "A Low-Noise Estimator of Angular Speed and Acceleration from Shaft Encoder Measurements"
(*
	THETA_ERR_FAST:=THETA_rads-THETA_EST_TOT;
	//  limit maybe to much lower than 2pi 
	
	IF abs(THETA_ERR_FAST) > THETA_ERR_HYS THEN
		OMEGA_FAST:= GAIN_EST*THETA_ERR_FAST;
		
	ELSE
 		OMEGA_FAST:=0;

	END_IF			
	

	OMEGA_EST_TOT:= OMEGA_filtered+OMEGA_FAST;
	THETA_EST_FAST := THETA_EST_FAST_OLD+ OMEGA_EST_TOT*Ts_EST;
	THETA_EST_TOT:=THETA_EST_FAST +0.5*Ts_EST*OMEGA_filtered;
	REST:=THETA_EST_TOT;
	
	 //IF THETA_EST_TOT >= 2*pi 
	IF THETA_EST_TOT < 0 THEN
		THETA_EST_TOT_OLD :=THETA_EST_TOT_OLD+2*PI;   
		THETA_EST_TOT := 2*PI+THETA_EST_TOT;// - (0 - THETA_EST_TOT) ;  
		THETA_EST_FAST_OLD :=THETA_EST_FAST_OLD+2*PI;   
		THETA_EST_FAST:= 2*PI+THETA_EST_FAST;
		
	//UNDERFLOW_SET := TRUE;
	
	ELSIF THETA_EST_TOT > 2*PI THEN
		THETA_EST_TOT_OLD :=THETA_EST_TOT_OLD-2*PI;   ;
		THETA_EST_TOT := THETA_EST_TOT-2*PI;// - (0 - THETA_EST_TOT) ;  
		THETA_EST_FAST_OLD :=0;//THETA_EST_FAST_OLD-2*PI;   
		THETA_EST_FAST:= 0;//THETA_EST_FAST-2*PI;
		//THETA_EST_TOT := 0;// + (THETA_EST_TOT - 2*PI) ;  //FOR THE SAME REASON
	//OVERFLOW_SET := TRUE;
	END_IF
		
		THETA_EST_FAST_OLD:= THETA_EST_FAST;
		THETA_EST_TOT_OLD := THETA_EST_TOT; 
	
	//end of fast speed estimator part
*)

//End of angular rotation speed estimation

//Rotor angle theta conversion deg -> rad and limitation
THETA := PI*THETA/180.0;
THETA_EL := PI*THETA_EL/180.0;

IF THETA < 0 THEN
	THETA := 0;
ELSIF
	THETA > 2*PI THEN
	THETA := 2*PI;
END_IF

IF THETA_EL < 0 THEN
	THETA_EL := 0;
ELSIF THETA_EL > 2*PI THEN
	THETA_EL := 2*PI;
END_IF

//End of rotor angle theta conversion deg->rad and limitation

END_FUNCTION_BLOCK

// ---- OLD/FB_Encoder_Old2.TcPOU
FUNCTION_BLOCK FB_Encoder_Old2
VAR CONSTANT
	nAmountOfSamples				: UINT := 100;
	fSamplingTime					: REAL := 0.00005; // 50us
	fCounterToRotationMultiplier	: REAL := 0.25; // Multiplier that transforms the counter value back to rotation.
	fMaxCounterIncrement			: REAL := 30000;
END_VAR
VAR
	nCounterValue 					: REFERENCE TO UINT; // Reference to value that holds the encoder value
	aPositionArray					: ARRAY [0..nAmountOfSamples-1] OF UINT; // Hold those positions in array.
	nValueCount						: UINT; // Rolling number used to store positions
	nStartCount						: UINT; // Value that holds the current starting value.
END_VAR

METHOD AddPosition : BOOL

IF nValueCount < nAmountOfSamples THEN // Fill samples
	aPositionArray[nValueCount] := nCounterValue;
	nStartCount := 0;
	nValueCount := nValueCount + 1;
ELSE // When all samples are full, move starting point forward by one. Write new value.
	nStartCount := nStartCount + 1;
	IF nStartCount = nAmountOfSamples THEN
		nStartCount := 0;
	END_IF
	
	IF nStartCount = 0 THEN
		aPositionArray[nValueCount] := nCounterValue;
	ELSE
		aPositionArray[nStartCount-1] := nCounterValue;
	END_IF
	
END_IF
END_METHOD

METHOD CalculateSpeed : REAL
VAR
	i,j 				: UINT;
	nUINTMax			: REAL := 16#FFFF;
	fTempRotationValueS	: REAL;
	fTempRotationValueE : REAL;
	fTempTotalRotation	: REAL := 0.0;
	fTempRotation		: REAL := 0.0;
	fTimeDuration		: REAL;
END_VAR
IF nValueCount < nAmountOfSamples THEN
	CalculateSpeed := 0;
ELSE
	CalculateSpeed := 0;
	fTimeDuration := fSamplingTime * nAmountOfSamples;
	FOR i := 0 TO nAmountOfSamples-1 DO
		j := nStartCount + i;
		IF j > nAmountOfSamples-1 THEN
			j := j-nAmountOfSamples;
		END_IF
		fTempRotationValueS	:= UINT_TO_REAL(aPositionArray[j]);
		
		IF j = nAmountOfSamples-1 THEN // If j value is at max index.
			fTempRotationValueE	:= UINT_TO_REAL(aPositionArray[0]);
		ELSE
			fTempRotationValueE	:= UINT_TO_REAL(aPositionArray[j+1]);
		END_IF
		
		fTempRotation := fTempRotationValueE - fTempRotationValueS; // The difference between starting point and the end point == Distance rotated between the cycles
		
		// Detection for counter overflow
		IF fTempRotation < -fMaxCounterIncrement THEN
			fTempRotation := fTempRotationValueE - fTempRotationValueS+nUINTMax;
		ELSIF fTempRotation > fMaxCounterIncrement THEN
			fTempRotation := fTempRotationValueE-nUINTMax - fTempRotationValueS;
		END_IF
		
		fTempTotalRotation := fTempTotalRotation + (fTempRotation * fCounterToRotationMultiplier);
	END_FOR
	CalculateSpeed := fTempTotalRotation/fTimeDuration; // Total Rotations during the measurement duration
	CalculateSpeed := CalculateSpeed * (60/fTimeDuration); // Multiplied to Rounds per minute
END_IF
END_METHOD

METHOD FB_init : BOOL
VAR_INPUT
	bInitRetains : BOOL; // if TRUE, the retain variables are initialized (warm start / cold start)
	bInCopyCode : BOOL;  // if TRUE, the instance afterwards gets moved into the copy code (online change)

	nCounter_In : REFERENCE TO UINT; // Reference to value that holds the encoder value.
END_VAR

nValueCount		:= 0; // There is currently no values in storage.
nCounterValue REF= nCounter_In; // Set the refence of counter value.
END_METHOD

END_FUNCTION_BLOCK

// ---- OLD/FB_Encoder_V2.TcPOU
FUNCTION_BLOCK FB_Encoder_V2
VAR_INPUT
END_VAR

VAR_OUTPUT
	THETA : REAL;
	THETA_EL : REAL;
	OMEGA: REAL;
END_VAR

VAR
	OMEGA_raw: REAL;
	OMEGA_filtered: REAL;
	Omega_prev: REAL;
	THETA_rads: REAL;
	THETA_prev_rads: REAL;
	
	THETA_PREV : REAL := 0;
	T_S : REAL := 0.0001;
	OVERFLOW_SET : BOOL := FALSE;
	UNDERFLOW_SET : BOOL := FALSE;

	UNDERFLOW_VALUE : UINT := 0;
	OVERFLOW_VALUE : UINT := 65535;
	DOWNCOUNT_VALUE : UINT := 1003;
	UPCOUNT_VALUE : UINT := DOWNCOUNT_VALUE + (PULSES_PER_REV - 1);
	
	INIT_DONE : BOOL := FALSE;
	
	I : INT := 0;
	COUNTER_VALUE_PREV : UINT := COUNTER_VALUE;
	COUNTER_OUT : UINT := 0;
	FIRSTCYCLE_DONE : BOOL := FALSE;
	CLOCKWISE: BOOL;
	COUNTERCLOCKWISE: BOOL;
	PLUSONEPULSE : BOOL;
	PLUSTWOPULSES :  BOOL;
	PLUSTHREEPULSES : BOOL;
	
	THETA_EST_TOT :REAL;
	THETA_EST_TOT_OLD: REAL:=0.0;
	THETA_ERR_FAST: REAL;
	THETA_ERR_HYS: REAL:= 0.1;//0.1
	OMEGA_FAST :REAL;
	OMEGA_EST_TOT :REAL;
	Ts_EST :REAL :=1E-4;//1E-2
	THETA_EST_FAST :REAL;
	THETA_EST_FAST_OLD :REAL;
	GAIN_EST :REAL :=20; //1
	
	THETA_n :REAL; 
	DELTA_THETA_n0 :REAL :=0.0;
	DELTA_THETA_n1 :REAL :=0.0; 
	DELTA_THETA :REAL; 
	
END_VAR


//Init procedure
IF FIRSTCYCLE_DONE = FALSE THEN
(*	STARTING_VALUE := COUNTER_VALUE;
	UP_VALUE := STARTING_VALUE + PULSES_PER_REV;
	DOWN_VALUE := STARTING_VALUE - PULSES_PER_REV;
*)	FIRSTCYCLE_DONE := TRUE;
END_IF

//End of init procedure

//Rotation direction estimation											//ADDED ROTATION  DIRECTION ESTIMATION - FEDOR POLUNIN 07 06 17

	IF (COUNTER_VALUE < COUNTER_VALUE_PREV AND COUNTER_VALUE <= (UNDERFLOW_VALUE + 2) AND COUNTER_VALUE_PREV >= (OVERFLOW_VALUE - 2)) THEN
		CLOCKWISE := TRUE;
		COUNTERCLOCKWISE := FALSE;
	ELSIF (COUNTER_VALUE > COUNTER_VALUE_PREV AND COUNTER_VALUE_PREV <= (UNDERFLOW_VALUE + 2) AND COUNTER_VALUE >= (OVERFLOW_VALUE - 2)) THEN
		COUNTERCLOCKWISE := TRUE;
		CLOCKWISE := FALSE;
	ELSIF 	(COUNTER_VALUE > COUNTER_VALUE_PREV AND COUNTER_VALUE <> OVERFLOW_VALUE) THEN 
		CLOCKWISE := TRUE;
		COUNTERCLOCKWISE := FALSE;
	ELSIF 	(COUNTER_VALUE < COUNTER_VALUE_PREV AND COUNTER_VALUE <> UNDERFLOW_VALUE) THEN
		COUNTERCLOCKWISE := TRUE;
		CLOCKWISE := FALSE;
	END_IF

//COUNTERCLOCKWISE := TRUE;
//CLOCKWISE := TRUE;

//End of Rotation direction estimation 

// Counter value conversion from 0..65535 to DOWNCOUNT_VALUE .. UPCOUNT_VALUE (1003..2002)  		//up to 1200 rpm both directions, no pulse loss w/o load Fedor Polunin 26 06 2017

IF (COUNTER_VALUE <= (UNDERFLOW_VALUE + 2) AND COUNTER_VALUE_PREV >= (OVERFLOW_VALUE - 2)) THEN
	COUNTER_OUT := COUNTER_OUT + (COUNTER_VALUE-UNDERFLOW_VALUE) + (OVERFLOW_VALUE-COUNTER_VALUE_PREV) + 1; 	//added + 1 because otherwise when COUNTER_VALUE resets from 65535 to 0, COUNTER_OUT does not increment
ELSIF (COUNTER_VALUE >= (OVERFLOW_VALUE - 2) AND COUNTER_VALUE_PREV <= (UNDERFLOW_VALUE + 2)) THEN
	COUNTER_OUT := COUNTER_OUT - (OVERFLOW_VALUE-COUNTER_VALUE) - (COUNTER_VALUE_PREV-UNDERFLOW_VALUE) - 1;		//added - 1 because otherwise when COUNTER_VALUE resets from 0 to 65535, COUNTER_OUT does not decrement
ELSIF (COUNTER_VALUE = COUNTER_VALUE_PREV + 1) OR (COUNTER_VALUE = COUNTER_VALUE_PREV + 2) OR (COUNTER_VALUE = COUNTER_VALUE_PREV + 3)THEN			
	COUNTER_OUT := COUNTER_OUT + (COUNTER_VALUE - COUNTER_VALUE_PREV); // + 1;
ELSIF  (COUNTER_VALUE = COUNTER_VALUE_PREV - 1) OR (COUNTER_VALUE = COUNTER_VALUE_PREV - 2) OR (COUNTER_VALUE = COUNTER_VALUE_PREV - 3) THEN; 
	COUNTER_OUT := COUNTER_OUT - (COUNTER_VALUE_PREV - COUNTER_VALUE);//- 1;
END_IF

IF COUNTER_OUT < DOWNCOUNT_VALUE THEN
	COUNTER_OUT := UPCOUNT_VALUE - (DOWNCOUNT_VALUE - COUNTER_OUT) + 1;  // +1 TO PREVENT COUNTER_OUT FROM SETTING UP TO 2001 INSTEAD OF 2002 WHEN DOWNCOUNT_VALUE - COUNTER_OUT = 1
	UNDERFLOW_SET := TRUE;
	
ELSIF COUNTER_OUT > UPCOUNT_VALUE THEN
	COUNTER_OUT := DOWNCOUNT_VALUE + (COUNTER_OUT - UPCOUNT_VALUE) - 1;  //FOR THE SAME REASON
	OVERFLOW_SET := TRUE;
END_IF

(*	
	//Encoder pulses per program cycle counter														
IF (COUNTER_VALUE = COUNTER_VALUE_PREV + 1) THEN
	PLUSONEPULSE := TRUE;
	PLUSTWOPULSES := FALSE;
	PLUSTHREEPULSES := FALSE;
	
ELSIF (COUNTER_VALUE = COUNTER_VALUE_PREV + 2) THEN
	PLUSONEPULSE := FALSE;
	PLUSTWOPULSES := TRUE;
	PLUSTHREEPULSES := FALSE;
	
ELSIF (COUNTER_VALUE = COUNTER_VALUE_PREV + 3) THEN
	PLUSONEPULSE := FALSE;
	PLUSTWOPULSES := FALSE;
	PLUSTHREEPULSES := TRUE;
END_IF
*)

COUNTER_VALUE_PREV := COUNTER_VALUE;

//End of counter value conversion 

// Convert to rotor angle theta in degrees

	THETA := 360.0*INT_TO_REAL(COUNTER_OUT - DOWNCOUNT_VALUE)/1000.0;		// COUNTER_OUT - DOWNCOUNT_VALUE can be negative, requires INT_TO_REAL 
    THETA_EL := 360.0*INT_TO_REAL(((COUNTER_OUT - DOWNCOUNT_VALUE) MOD 200))/200.0;

//End of conversion to rotor angle theta in degrees

//Angular rotation speed omega estimation (in rad/s)
I := I+1;

	THETA_rads := THETA*PI/180;

IF I = SPEED_CALC_Cycle THEN															
	// Calculate angular speed
		//raw speed estimation algorithm based on backward Euler differentiation
	IF OVERFLOW_SET = TRUE AND THETA < 20 THEN								//Fedor Polunin 06.06.17 - added AND THETA < 10 to prevent this from executing if theta hasn't yet changed from 2pi to zero
		OMEGA := (THETA + (360.0 - THETA_PREV))/(T_S*SPEED_CALC_Cycle);				
	ELSIF UNDERFLOW_SET = TRUE AND THETA > 340 THEN							//Fedor Polunin 06.06.17 - added AND THETA < 10 to prevent this from executing if theta hasn't yet changed from zero to 2pi
		OMEGA := -((360.0-THETA) + THETA_PREV)/(T_S*SPEED_CALC_Cycle);					
	ELSE
		IF CLOCKWISE = TRUE AND THETA_PREV > 180 AND THETA < 180 THEN		//Fedor Polunin 06.06.17 - added                                                                                           (IF THETA_PREV > 180 AND THETA < 180 THEN) BUT NOT VALID if both directions are used (it is to ensure correct omega estimation during THETA 2pi to 0 change)
			OMEGA := (THETA + (360.0 - THETA_PREV))/(T_S*SPEED_CALC_Cycle);			//Fedor Polunin 06.06.17 - added OMEGA := (THETA + (360.0 - THETA_PREV))/(T_S*100.0);
		ELSIF  COUNTERCLOCKWISE = TRUE AND  THETA_PREV < 180 AND THETA > 180 THEN							
			OMEGA := -((360.0-THETA) + THETA_PREV)/(T_S*SPEED_CALC_Cycle);			
		ELSE																//Fedor Polunin 06.06.17 - ELSE use theta and theta_prev without modification:
			OMEGA := (THETA - THETA_PREV)/(T_S*SPEED_CALC_Cycle);
		END_IF
	END_IF	
	
	OMEGA_raw := PI*OMEGA/180.0;
	
	//end of raw speed estimation algorithm														
	
	//filtered speed estimation algorithm based on ZOH differentiation + filter + output median filtering		
	IF OVERFLOW_SET = TRUE AND THETA < 20 THEN								//Fedor Polunin 06.06.17 - added AND THETA < 10 to prevent this from executing if theta hasn't yet changed from 2pi to zero
		DELTA_THETA := (THETA_rads + (2*PI - THETA_prev_rads));		
	ELSIF UNDERFLOW_SET = TRUE AND THETA > 340 THEN							//Fedor Polunin 06.06.17 - added AND THETA < 10 to prevent this from executing if theta hasn't yet changed from zero to 2pi
		DELTA_THETA := -((2*PI-THETA_rads ) + THETA_prev_rads);				
	ELSE
		IF CLOCKWISE = TRUE AND THETA_PREV > 180 AND THETA < 180 THEN		//Fedor Polunin 06.06.17 - added                                                                                           (IF THETA_PREV > 180 AND THETA < 180 THEN) BUT NOT VALID if both directions are used (it is to ensure correct omega estimation during THETA 2pi to 0 change)
			DELTA_THETA := (THETA_rads  + (2*PI - THETA_prev_rads));				//Fedor Polunin 06.06.17 - added OMEGA := (THETA + (360.0 - THETA_PREV))/(T_S*100.0);
		ELSIF  COUNTERCLOCKWISE = TRUE AND  THETA_PREV < 180 AND THETA > 180 THEN							
			DELTA_THETA := -((2*PI-THETA_rads ) + THETA_prev_rads);	
		ELSE																//Fedor Polunin 06.06.17 - ELSE use theta and theta_prev without modification:
			DELTA_THETA := (THETA_rads  - THETA_prev_rads);	
		END_IF
	END_IF														
	
	DELTA_THETA_n0:=0.5*DELTA_THETA+ 0.5*DELTA_THETA_n1;
 	DELTA_THETA_n1:= DELTA_THETA_n0;
	OMEGA_filtered := DELTA_THETA_n0*33*104.0166/21.23 +  0.189 * Omega_prev ;	

	THETA_PREV := THETA;
	THETA_prev_rads := THETA_rads;
	OMEGA_prev:= OMEGA_filtered;
	
	//end of filtered speed estimation algorithm
	
	I := 0;

	UNDERFLOW_SET := FALSE;
	OVERFLOW_SET := FALSE;
	
	//Speed feedback signal selection
		//OMEGA:=OMEGA_raw;
		OMEGA:=OMEGA_filtered;
END_IF;
	
	//fast speed estimator part (filtered algorithm above is the slow part) - refer to the paper "A Low-Noise Estimator of Angular Speed and Acceleration from Shaft Encoder Measurements"
(*
	THETA_ERR_FAST:=THETA_rads-THETA_EST_TOT;
	//  limit maybe to much lower than 2pi 
	
	IF abs(THETA_ERR_FAST) > THETA_ERR_HYS THEN
		OMEGA_FAST:= GAIN_EST*THETA_ERR_FAST;
		
	ELSE
 		OMEGA_FAST:=0;

	END_IF			
	

	OMEGA_EST_TOT:= OMEGA_filtered+OMEGA_FAST;
	THETA_EST_FAST := THETA_EST_FAST_OLD+ OMEGA_EST_TOT*Ts_EST;
	THETA_EST_TOT:=THETA_EST_FAST +0.5*Ts_EST*OMEGA_filtered;
	REST:=THETA_EST_TOT;
	
	 //IF THETA_EST_TOT >= 2*pi 
	IF THETA_EST_TOT < 0 THEN
		THETA_EST_TOT_OLD :=THETA_EST_TOT_OLD+2*PI;   
		THETA_EST_TOT := 2*PI+THETA_EST_TOT;// - (0 - THETA_EST_TOT) ;  
		THETA_EST_FAST_OLD :=THETA_EST_FAST_OLD+2*PI;   
		THETA_EST_FAST:= 2*PI+THETA_EST_FAST;
		
	//UNDERFLOW_SET := TRUE;
	
	ELSIF THETA_EST_TOT > 2*PI THEN
		THETA_EST_TOT_OLD :=THETA_EST_TOT_OLD-2*PI;   ;
		THETA_EST_TOT := THETA_EST_TOT-2*PI;// - (0 - THETA_EST_TOT) ;  
		THETA_EST_FAST_OLD :=0;//THETA_EST_FAST_OLD-2*PI;   
		THETA_EST_FAST:= 0;//THETA_EST_FAST-2*PI;
		//THETA_EST_TOT := 0;// + (THETA_EST_TOT - 2*PI) ;  //FOR THE SAME REASON
	//OVERFLOW_SET := TRUE;
	END_IF
		
		THETA_EST_FAST_OLD:= THETA_EST_FAST;
		THETA_EST_TOT_OLD := THETA_EST_TOT; 
	
	//end of fast speed estimator part
*)

//End of angular rotation speed estimation

//Rotor angle theta conversion deg -> rad and limitation
THETA := PI*THETA/180.0;
THETA_EL := PI*THETA_EL/180.0;

IF THETA < 0 THEN
	THETA := 0;
ELSIF
	THETA > 2*PI THEN
	THETA := 2*PI;
END_IF

IF THETA_EL < 0 THEN
	THETA_EL := 0;
ELSIF THETA_EL > 2*PI THEN
	THETA_EL := 2*PI;
END_IF

//End of rotor angle theta conversion deg->rad and limitation

END_FUNCTION_BLOCK

// ---- OLD/FB_ENCODER_V3.TcPOU
FUNCTION_BLOCK FB_ENCODER_V3
VAR_OUTPUT
	THETA_EL 			: REAL;
	THETA_MECH 			: REAL;
	OMEGA_EL 			: REAL;
	OMEGA_MECH 			: REAL;
END_VAR
VAR
	COUNTER_MAX 		: UINT := 16383;
	COUNTER_INV_MAX 	: UINT := 65535;
	COUNTER_TEMP 		: UINT;
	SAMPLE_TIME			: REAL := 100E-6;
END_VAR
VAR_STAT
   	THETA_MECH_PREV 	: REAL := 0;
END_VAR


// If counter is maximum UINT value (or over COUNTER_MAX), rotation is reversed.
IF Measurements.COUNTER_VALUE > COUNTER_MAX THEN
	COUNTER_TEMP := COUNTER_MAX + (Measurements.COUNTER_VALUE - COUNTER_INV_MAX);
ELSE
	COUNTER_TEMP := Measurements.COUNTER_VALUE;
END_IF

IF Measurements.COUNTER_VALUE >= Measurements.COUNTER_OFFSET THEN
	COUNTER_TEMP := COUNTER_TEMP - Measurements.COUNTER_OFFSET;
ELSIF Measurements.COUNTER_VALUE < Measurements.COUNTER_OFFSET THEN
	COUNTER_TEMP := COUNTER_TEMP + Measurements.COUNTER_OFFSET;
END_IF

IF COUNTER_TEMP > COUNTER_MAX THEN
	COUNTER_TEMP := COUNTER_MAX;
END_IF

THETA_MECH := LREAL_TO_REAL(2*PI*UINT_TO_LREAL(COUNTER_TEMP)/UINT_TO_LREAL(COUNTER_MAX));

IF THETA_MECH*2 > 2*PI THEN
	THETA_EL := LREAL_TO_REAL(THETA_MECH*2 - 2*PI);
ELSE
	THETA_EL := THETA_MECH*2;
END_IF

OMEGA_MECH := (THETA_MECH-THETA_MECH_PREV)/SAMPLE_TIME;
THETA_MECH_PREV := THETA_MECH;

OMEGA_EL := OMEGA_MECH*2;

END_FUNCTION_BLOCK

// ---- OLD/FB_HomingTimer.TcPOU
FUNCTION_BLOCK FB_HomingTimer
VAR_OUTPUT
	bDone : BOOL;
END_VAR
VAR
	i			: LINT := 0;
	uLoopCount	: LINT;
END_VAR


bDone := FALSE;

i := i + 1;

IF i >= uLoopCount THEN
	bDone := TRUE;
END_IF

METHOD FB_init : BOOL
VAR_INPUT
	bInitRetains	: BOOL; // if TRUE, the retain variables are initialized (warm start / cold start)
	bInCopyCode		: BOOL;  // if TRUE, the instance afterwards gets moved into the copy code (online change)
	
	uLoopsToRun		: LINT;
END_VAR

THIS^.i := 0;
THIS^.uLoopCount := uLoopsToRun;
END_METHOD

END_FUNCTION_BLOCK

// ---- OLD/F_GenerateCANMessage.TcPOU
FUNCTION F_GenerateCANMessage : CANQUEUE
VAR_INPUT
	cobID	: UINT;
	V_a		: WORD;
	V_b		: WORD;
END_VAR
VAR
	i,j 		: UINT;
	Tempdata	: USINT;
	V_DWORD		: WORD;
	tempMessage : CANMESSAGE;
END_VAR


// WIP CAN Message writing.
(*
	Viestiin tulee Va ja Vb (ilmeisesti). Yksi CAN Frame on käytössä näille kahdelle muuttujalle.
	CANQUEUE Objekti on yksi CAN viesti, joka lähetetään COB ID:seen ja se sisältää 8 kpl UINT muuttujia, jotka varmaankin kirjoitetaan sarjassa, josta muodostuu se 64 bittinen CAN Frame.
	Ei kyllä ole kamalasti ideaa että missä järjestyksessä ne kirjoitetaan sinne. Eli pitäisi varmaankin testata. 
	Koodi on nyt silleensä että oletetaan että kirjoitetaan 7 -> 0. Jolloin 7:n data yksikön merkitsevin bitti on koko framen merkisevin
	Vastaavasti 0:n viimeinen bitti on koko framen viimeinen kirjoitettava bitti.
*)


F_GenerateCANMessage.cobId := cobID;

V_DWORD := V_a;
FOR j := 0 TO 1 DO // First part of frame reserved for V_a
	CASE j OF // ST is dumb language and doesnt allow looping for bit access.
		1:
			Tempdata.0 := V_DWORD.0;
			Tempdata.1 := V_DWORD.1;
			Tempdata.2 := V_DWORD.2;
			Tempdata.3 := V_DWORD.3;
			Tempdata.4 := V_DWORD.4;
			Tempdata.5 := V_DWORD.5;
			Tempdata.6 := V_DWORD.6;
			Tempdata.7 := V_DWORD.7;
			
		0:
			Tempdata.0 := V_DWORD.8;
			Tempdata.1 := V_DWORD.9;
			Tempdata.2 := V_DWORD.10;
			Tempdata.3 := V_DWORD.11;
			Tempdata.4 := V_DWORD.12;
			Tempdata.5 := V_DWORD.13;
			Tempdata.6 := V_DWORD.14;
			Tempdata.7 := V_DWORD.15;
	ELSE
		RETURN;
	END_CASE
	F_GenerateCANMessage.data[j] := Tempdata;
END_FOR

V_DWORD := V_b;
FOR j := 2 TO 3 DO // Second part is reserved for V_b
	CASE j OF // ST is dumb language and doesnt allow looping for bit access.
		3:
			Tempdata.0 := V_DWORD.0;
			Tempdata.1 := V_DWORD.1;
			Tempdata.2 := V_DWORD.2;
			Tempdata.3 := V_DWORD.3;
			Tempdata.4 := V_DWORD.4;
			Tempdata.5 := V_DWORD.5;
			Tempdata.6 := V_DWORD.6;
			Tempdata.7 := V_DWORD.7;
			
		2:
			Tempdata.0 := V_DWORD.8;
			Tempdata.1 := V_DWORD.9;
			Tempdata.2 := V_DWORD.10;
			Tempdata.3 := V_DWORD.11;
			Tempdata.4 := V_DWORD.12;
			Tempdata.5 := V_DWORD.13;
			Tempdata.6 := V_DWORD.14;
			Tempdata.7 := V_DWORD.15;
	ELSE
		RETURN;
	END_CASE
	F_GenerateCANMessage.data[j] := Tempdata;
END_FOR

END_FUNCTION

// ---- OLD/F_Homing.TcPOU
FUNCTION F_Homing : BOOL
VAR
	LoopCount	: INT := 2000;
END_VAR

END_FUNCTION

// ---- OLD/F_MechToEl.TcPOU
FUNCTION F_MechToEl : LREAL
VAR_INPUT
	w_mech : LREAL;
	p : 	LREAL;
END_VAR
VAR
	w_el : LREAL;
END_VAR


w_el := w_mech * p;

IF w_el > 2*PI THEN
	w_el := w_el - 2*pi;
END_IF

F_MechToEl := w_el;

END_FUNCTION

// ---- OLD/F_VoltageToWord.TcPOU
FUNCTION F_VoltageToWord : WORD
VAR_INPUT
	Voltage_In			: REAL; // Voltage input
END_VAR
VAR
	VoltageMultiplier	: REAL;
	MaxWordValue		: REAL := 16#FFFF;
	Voltage_High_Value 	: REAL := 0.866;
	Voltage_Low_Value	: REAL := -0.866;
END_VAR

// Check that voltage value is between min and max value.
IF Voltage_In > Voltage_High_Value THEN
	Voltage_In := Voltage_High_Value;
ELSIF Voltage_In < Voltage_Low_Value THEN
	Voltage_In := Voltage_Low_Value;
END_IF

VoltageMultiplier := (Voltage_In-Voltage_Low_Value)/(Voltage_High_Value-Voltage_Low_Value);

F_VoltageToWord := UINT_TO_WORD(REAL_TO_UINT(VoltageMultiplier*MaxWordValue));

END_FUNCTION

// ---- POUs/F_AnalogIntToVoltage.TcPOU
FUNCTION F_AnalogIntToVoltage : REAL
VAR_INPUT
	AnalogValue	: INT;
END_VAR
VAR
	Max_Int_Value_pos	: INT := 32767;
	Max_Int_Value_Neg	: INT := -32768;
	Voltagevalue 		: REAL := 10;
END_VAR



IF AnalogValue > 0 THEN
	F_AnalogIntToVoltage := Voltagevalue*(INT_TO_REAL(AnalogValue)/INT_TO_REAL(Max_Int_Value_pos));
ELSIF AnalogValue < 0 THEN
	F_AnalogIntToVoltage :=  Voltagevalue*(INT_TO_REAL(AnalogValue)/INT_TO_REAL(Max_Int_Value_Neg));
ELSE
	F_AnalogIntToVoltage := 0;
END_IF

END_FUNCTION

// ---- POUs/F_VoltageToCurrentConvert.TcPOU
FUNCTION F_VoltageToCurrentConvert : REAL
VAR_INPUT
	VoltageValue 	: REAL;
END_VAR
VAR
	Current			: REAL;
	Gain			: REAL := 3.1809;
	Offset			: REAL := -7.933;
END_VAR

Current := VoltageValue*Gain + Offset;

F_VoltageToCurrentConvert := Current;

END_FUNCTION

// ---- GlobalTextList.TcGTLO
TEXTLIST GlobalTextList
  11 = 'CurrentMeasurement Value [V]'
  666 = 'Encoder Speed'
  841 = 'Encoder Speed [RPM]'
END_TEXTLIST

// ---- VISUs/Visualization.TcVIS
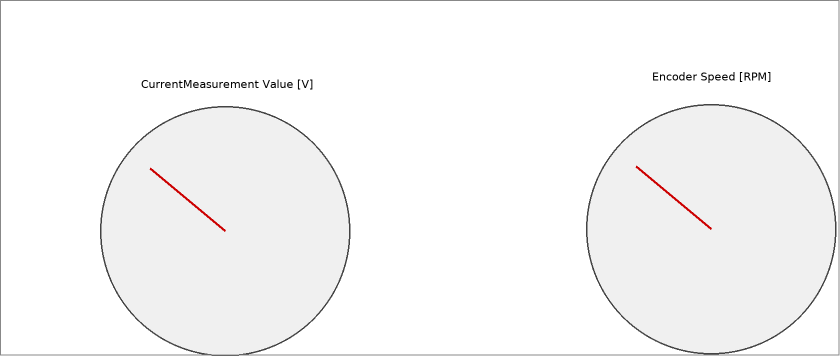
VISUALIZATION Visualization  // 840x356
    Meter180 (100,106 250x250), value: MAIN.CurrentMeasurement, style: Meter-Meter180-Gray, scale format: %.1f, scale -5..5
    Label (118,57 219x55), "CurrentMeasurement Value [V]"
    Meter180 (586,104 250x250), value: MAIN.CurrentMeasurement, style: Meter-Meter180-Gray, scale format: %.1f, scale 0..1000
    Label (584,47 256x60), "Encoder Speed [RPM]"
END_VISUALIZATION
